(* PLC project io_single_acting_jack, Dassault Systèmes ControlBuild 2024x *)
(* stored: creationDateTime 2023-10-03T11:12:48-01:00 *)

PROGRAM panel
  VAR_OUTPUT
    valveWorkPB : BOOL := false;
  END_VAR

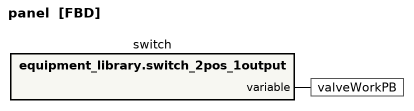
(* FBD diagram, written out as Structured Text *)
switch();
valveWorkPB := switch.variable;
END_PROGRAM

(* Integrated object C/C+OP of a single acting jack *)
PROGRAM io_library.io_single_acting_jack
  VAR_INPUT
    acknowledgePB : BOOL := false;
  END_VAR
  VAR_INPUT
    autoMode : BOOL := false;
    manualMode : BOOL := false;
  END_VAR
  VAR_INPUT
    autoWorkCmd : BOOL := false;
  END_VAR
  VAR_OUTPUT
    generalFault : BOOL := false;
  END_VAR
  VAR_OUTPUT
    inletSensor : BOOL := false;
    outletSensor : BOOL := false;
  END_VAR
  VAR_OUTPUT
    rodPosition : REAL := 0.0;
    rodPercent : REAL := 0.0;
    incrementValue : REAL := 0.0;
  END_VAR

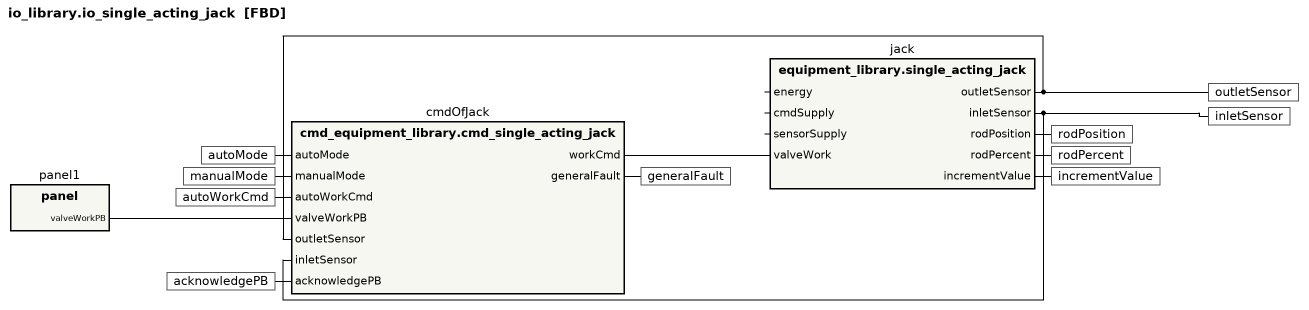
(* FBD diagram, written out as Structured Text *)
panel1();
jack(valveWork := cmdOfJack.workCmd);
cmdOfJack(autoMode := autoMode, manualMode := manualMode, autoWorkCmd := autoWorkCmd, valveWorkPB := panel1.valveWorkPB, outletSensor := jack.outletSensor, inletSensor := jack.inletSensor, acknowledgePB := acknowledgePB);
generalFault := cmdOfJack.generalFault;
inletSensor := jack.inletSensor;
outletSensor := jack.outletSensor;
rodPosition := jack.rodPosition;
rodPercent := jack.rodPercent;
incrementValue := jack.incrementValue;
END_PROGRAM
